Omron CX-Programmer project NewProject (CX-Programmer 9.61)

# PLC Mod_2_1: CP1H XA

## Global symbols (name address type ; comment)
200 CHANNEL  ; Temperature Sensor Analog Input
210 CHANNEL  ; VFD Frequency Reference Output Channel
D10 CHANNEL  ; Temperature Input (0-1.5V) in Analog Resolution
D15 CHANNEL  ; BCD Equivalent of Temperature Input
D20 CHANNEL  ; VFD Frequency Reference Output
D25 CHANNEL  ; BCD Equivalent of Voltage Supplied to VFD Frequency Reference
T0000 BOOL  ; Initialization Delay

## Program PLC__Temperature_Sensor__and_VFD_Controlled_Fan (cyclic task 0)
Local symbols
HIGH 32.00 BOOL  ; 32.00 - HIGH
HMI_VFD_MA 10.00 BOOL  ; 10.00 - HMI_VFD_MA
HMI_VFD_S1 10.01 BOOL  ; 10.01 - HMI_VFD_S1
HMI_VFD_S2 10.02 BOOL  ; 10.02 - HMI_VFD_S2
HMI_VFD_S3 10.03 BOOL  ; 10.03 - HMI_VFD_S3
HMI_VFD_S4 10.04 BOOL  ; 10.04 - HMI_VFD_S4
HMI_VFD_S5 10.05 BOOL  ; 10.05 - HMI_VFD_S5
LOW 30.00 BOOL  ; 30.00 - LOW
MEDIUM 31.00 BOOL  ; 31.00 - MEDIUM
PB_VFD_S1 0.01 BOOL  ; 0.01 - PB_VFD_S1
PB_VFD_S2 0.02 BOOL  ; 0.02 - PB_VFD_S2
PB_VFD_S3 0.03 BOOL  ; 0.03 - PB_VFD_S3
PB_VFD_S4 0.04 BOOL  ; 0.04 - PB_VFD_S4
PB_VFD_S5 0.05 BOOL  ; 0.05 - PB_VFD_S5
VFD_MA 0.00 BOOL  ; 0.00 - VFD_MA
VFD_S1 100.00 BOOL  ; 100.00 - VFD_S1
VFD_S2 100.04 BOOL  ; 100.04 - VFD_S2
VFD_S3 100.05 BOOL  ; 100.05 - VFD_S3
VFD_S4 100.06 BOOL  ; 100.06 - VFD_S4
VFD_S5 100.07 BOOL  ; 100.07 - VFD_S5

### Section Initialization

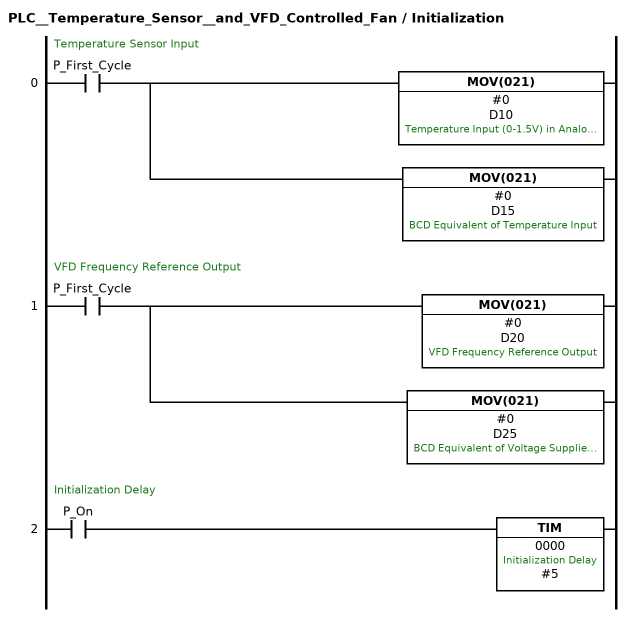
; rung 0: Temperature Sensor Input
LD P_First_Cycle
MOV(021) #0 D10  ; Temperature Input (0-1.5V) in Analog Resolution
MOV(021) #0 D15  ; BCD Equivalent of Temperature Input
; rung 1: VFD Frequency Reference Output
LD P_First_Cycle
MOV(021) #0 D20  ; VFD Frequency Reference Output
MOV(021) #0 D25  ; BCD Equivalent of Voltage Supplied to VFD Frequency Reference
; rung 2: Initialization Delay
LD P_On
TIM 0000 #5  ; Initialization Delay

### Section Main_Program

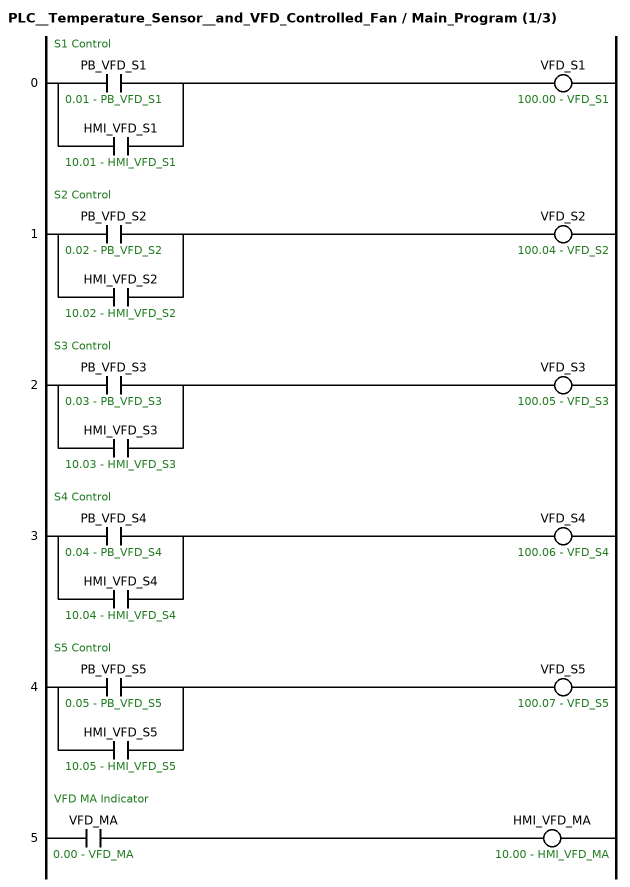
; rung 0: S1 Control
LD PB_VFD_S1  ; 0.01 - PB_VFD_S1
OR HMI_VFD_S1  ; 10.01 - HMI_VFD_S1
OUT VFD_S1  ; 100.00 - VFD_S1
; rung 1: S2 Control
LD PB_VFD_S2  ; 0.02 - PB_VFD_S2
OR HMI_VFD_S2  ; 10.02 - HMI_VFD_S2
OUT VFD_S2  ; 100.04 - VFD_S2
; rung 2: S3 Control
LD PB_VFD_S3  ; 0.03 - PB_VFD_S3
OR HMI_VFD_S3  ; 10.03 - HMI_VFD_S3
OUT VFD_S3  ; 100.05 - VFD_S3
; rung 3: S4 Control
LD PB_VFD_S4  ; 0.04 - PB_VFD_S4
OR HMI_VFD_S4  ; 10.04 - HMI_VFD_S4
OUT VFD_S4  ; 100.06 - VFD_S4
; rung 4: S5 Control
LD PB_VFD_S5  ; 0.05 - PB_VFD_S5
OR HMI_VFD_S5  ; 10.05 - HMI_VFD_S5
OUT VFD_S5  ; 100.07 - VFD_S5
; rung 5: VFD MA Indicator
LD VFD_MA  ; 0.00 - VFD_MA
OUT HMI_VFD_MA  ; 10.00 - HMI_VFD_MA

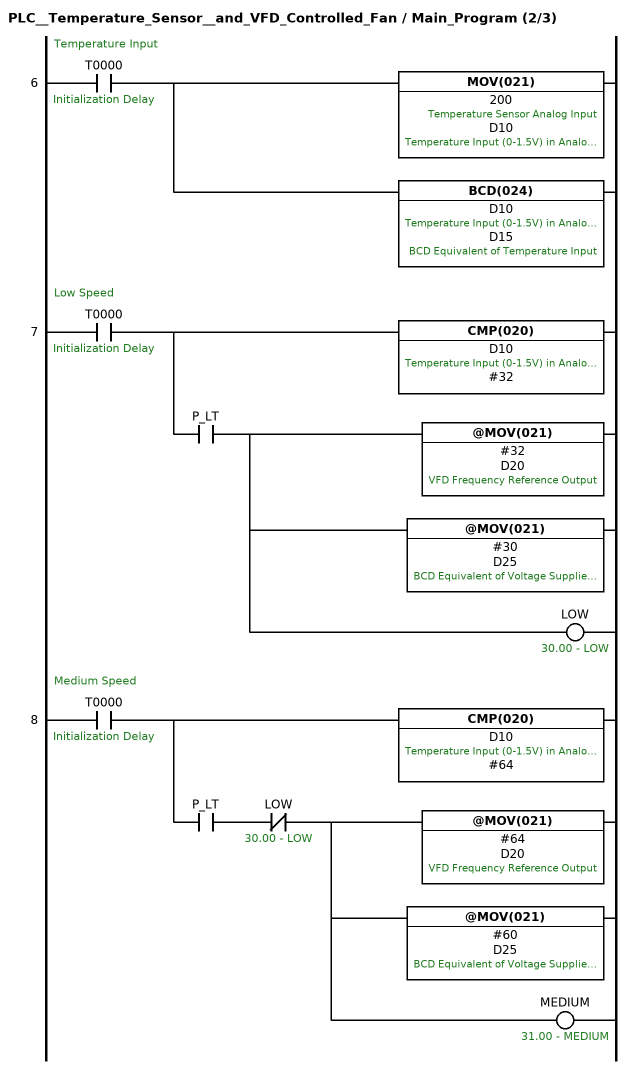
; rung 6: Temperature Input
LD T0000  ; Initialization Delay
MOV(021) 200 D10  ; Temperature Sensor Analog Input, Temperature Input (0-1.5V) in Analog Resolution
BCD(024) D10 D15  ; Temperature Input (0-1.5V) in Analog Resolution, BCD Equivalent of Temperature Input
; rung 7: Low Speed
LD T0000  ; Initialization Delay
CMP(020) D10 #32  ; Temperature Input (0-1.5V) in Analog Resolution
AND P_LT
@MOV(021) #32 D20  ; VFD Frequency Reference Output
@MOV(021) #30 D25  ; BCD Equivalent of Voltage Supplied to VFD Frequency Reference
OUT LOW  ; 30.00 - LOW
; rung 8: Medium Speed
LD T0000  ; Initialization Delay
CMP(020) D10 #64  ; Temperature Input (0-1.5V) in Analog Resolution
AND P_LT
ANDNOT LOW  ; 30.00 - LOW
@MOV(021) #64 D20  ; VFD Frequency Reference Output
@MOV(021) #60 D25  ; BCD Equivalent of Voltage Supplied to VFD Frequency Reference
OUT MEDIUM  ; 31.00 - MEDIUM

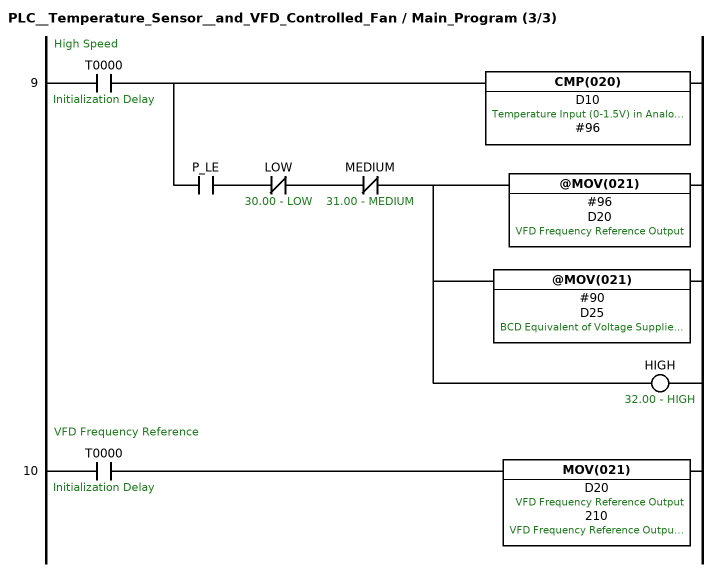
; rung 9: High Speed
LD T0000  ; Initialization Delay
CMP(020) D10 #96  ; Temperature Input (0-1.5V) in Analog Resolution
AND P_LE
ANDNOT LOW  ; 30.00 - LOW
ANDNOT MEDIUM  ; 31.00 - MEDIUM
@MOV(021) #96 D20  ; VFD Frequency Reference Output
@MOV(021) #90 D25  ; BCD Equivalent of Voltage Supplied to VFD Frequency Reference
OUT HIGH  ; 32.00 - HIGH
; rung 10: VFD Frequency Reference
LD T0000  ; Initialization Delay
MOV(021) D20 210  ; VFD Frequency Reference Output, VFD Frequency Reference Output Channel

### Section END
; rung 0
END(001)